// TIA Portal V19 export
FUNCTION_BLOCK "ForceNormalStop"   // FB8, F_LAD
// stored: Access Published
   VAR_INPUT
      Door_NormalStop : Bool;
      Door_SafeStop : Bool;
      AreaCycleOn : Bool;
   END_VAR
   VAR_OUTPUT
      ForceNormalStop : Bool;
   END_VAR
   VAR
      DlyRestartAfterDoorOpn : TON;
      MemDoorOpen : Bool;
      MemDoorsNewClosed : Bool;
   END_VAR
BEGIN

REGION Network 1: Froce Normal Stop
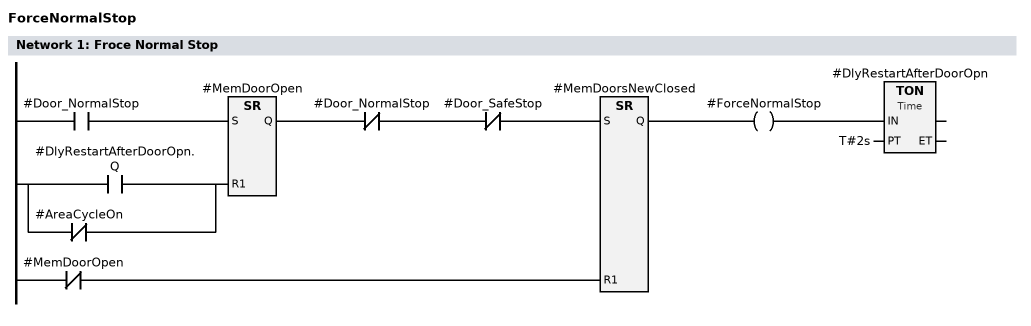
   RUNG wire#powerrail
      Contact( #Door_NormalStop )
      S_SR(operand := #MemDoorOpen, r1 := wire#w1)
      I_Contact( #Door_NormalStop )
      I_Contact( #Door_SafeStop )
      S_SR(operand := #MemDoorsNewClosed, r1 := wire#w2)
      Coil( #ForceNormalStop )
      { S7_Templates := "[time_type := Time, codedbool_type := DInt]" } #DlyRestartAfterDoorOpn.TON(pt := T#2s, et =>)
   END_RUNG
   RUNG wire#powerrail
      Contact( #DlyRestartAfterDoorOpn.Q )
   END_RUNG wire#w1
   RUNG wire#powerrail
      I_Contact( #AreaCycleOn )
   END_RUNG wire#w1
   RUNG wire#powerrail
      I_Contact( #MemDoorOpen )
   END_RUNG wire#w2
   // the same network as SCL:
   IF #Door_NormalStop THEN
       #MemDoorOpen := TRUE;   // SR flip-flop
   END_IF;
   IF #DlyRestartAfterDoorOpn.Q OR NOT #AreaCycleOn THEN #MemDoorOpen := FALSE; END_IF;
   IF #MemDoorOpen AND NOT #Door_NormalStop AND NOT #Door_SafeStop THEN
       #MemDoorsNewClosed := TRUE;   // SR flip-flop
   END_IF;
   IF NOT #MemDoorOpen THEN #MemDoorsNewClosed := FALSE; END_IF;
   #ForceNormalStop := #MemDoorsNewClosed;
   #DlyRestartAfterDoorOpn.TON(IN := #MemDoorsNewClosed, PT := T#2s);
END_REGION
END_FUNCTION_BLOCK
